FUNCTION_BLOCK StateMachine
VAR_INPUT
END_VAR
VAR_OUTPUT
END_VAR
VAR
	i : INT;
	State : States;
	TimerRotateDisc : TON;
	TimerLinearFW : TON;
	TimerGripperLower : TON;
	TimerGripperOpen : TON;
	TimerGripperClose: TON;
	TimerGripperLift: TON;
	TimerLinearBW : TON;
	Start: BOOL:=FALSE;
	CyclesCounter: CTU;
	TotalCyclesCounter : INT:=0;
	Reset : BOOL;
	NumberOfSlots : INT := 6;
	CylinderInDisc : ARRAY[1..6] OF BOOL := [FALSE, TRUE, TRUE, TRUE, TRUE, TRUE] ;
	Sensor: BOOL:= CylinderInDisc[4];
	PutCylinderInSlot6 : BOOL;
END_VAR

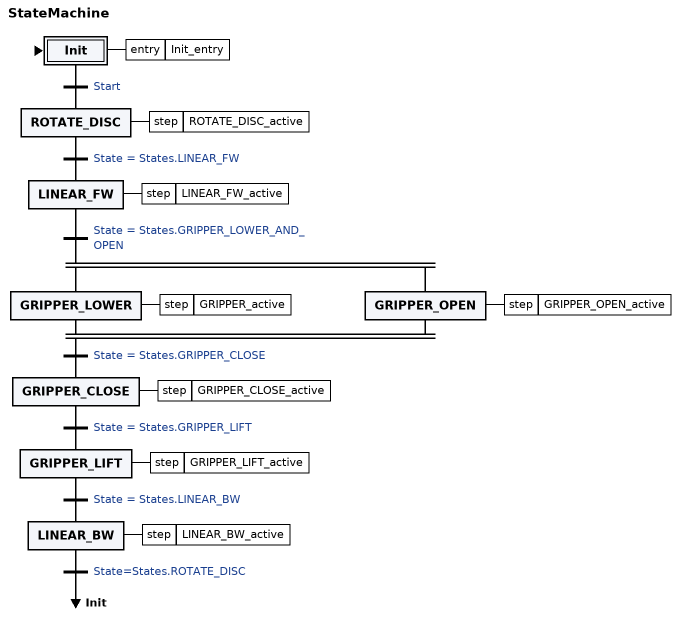
INITIAL_STEP Init:
    Init_entry(P1);  // entry action
END_STEP
TRANSITION FROM Init TO ROTATE_DISC
    := Start;
END_TRANSITION
STEP ROTATE_DISC:
    ROTATE_DISC_active(N);  // step action
END_STEP
TRANSITION FROM ROTATE_DISC TO LINEAR_FW
    := State = States.LINEAR_FW;
END_TRANSITION
STEP LINEAR_FW:
    LINEAR_FW_active(N);  // step action
END_STEP
TRANSITION FROM LINEAR_FW TO (GRIPPER_LOWER, GRIPPER_OPEN)
    := State = States.GRIPPER_LOWER_AND_OPEN;
END_TRANSITION
STEP GRIPPER_LOWER:
    GRIPPER_active(N);  // step action
END_STEP
STEP GRIPPER_OPEN:
    GRIPPER_OPEN_active(N);  // step action
END_STEP
TRANSITION FROM (GRIPPER_LOWER, GRIPPER_OPEN) TO GRIPPER_CLOSE
    := State = States.GRIPPER_CLOSE;
END_TRANSITION
STEP GRIPPER_CLOSE:
    GRIPPER_CLOSE_active(N);  // step action
END_STEP
TRANSITION FROM GRIPPER_CLOSE TO GRIPPER_LIFT
    := State = States.GRIPPER_LIFT;
END_TRANSITION
STEP GRIPPER_LIFT:
    GRIPPER_LIFT_active(N);  // step action
END_STEP
TRANSITION FROM GRIPPER_LIFT TO LINEAR_BW
    := State = States.LINEAR_BW;
END_TRANSITION
STEP LINEAR_BW:
    LINEAR_BW_active(N);  // step action
END_STEP
TRANSITION FROM LINEAR_BW TO Init
    := State=States.ROTATE_DISC;
END_TRANSITION

ACTION GRIPPER_active:
TimerGripperLower(IN:=TRUE, PT:=T#5S);
IF TimerGripperLower.Q THEN
	State := States.GRIPPER_CLOSE;
END_IF
END_ACTION

ACTION GRIPPER_CLOSE_active:
TimerGripperClose(IN:=TRUE, PT:=T#1S);
IF TimerGripperClose.Q THEN
	State := States.GRIPPER_LIFT;
END_IF
END_ACTION

ACTION GRIPPER_LIFT_active:
TimerGripperLift(IN:=TRUE, PT:=T#5S);
IF TimerGripperLift.Q THEN
	CylinderInDisc[1] := FALSE;
	State := States.LINEAR_BW;
END_IF
END_ACTION

ACTION GRIPPER_OPEN_active:
TimerGripperOpen(IN:=TRUE, PT:=T#1S);
END_ACTION

ACTION Init_entry:
Sensor := CylinderInDisc[4];

TimerRotateDisc(IN:=FALSE);
TimerLinearFW(IN:=FALSE);
TimerGripperLower(IN:=FALSE);
TimerGripperOpen(IN:=FALSE);
TimerGripperClose(IN:=FALSE);
TimerGripperLift(IN:=FALSE);
TimerLinearBW(IN:=FALSE);
Reset := CyclesCounter.Q;
CyclesCounter(CU:=state = States.ROTATE_DISC, RESET := Reset, PV:=INT_TO_WORD(NumberOfSlots));
END_ACTION

ACTION LINEAR_BW_active:
TimerLinearBW(IN:=TRUE, PT:=T#2S);
IF TimerLinearBW.Q THEN
	State := States.ROTATE_DISC;
END_IF
END_ACTION

ACTION LINEAR_FW_active:
TimerLinearFW(IN:=TRUE, PT:=T#2S);
IF TimerLinearFW.Q THEN
	State := States.GRIPPER_LOWER_AND_OPEN;
END_IF
END_ACTION

ACTION ROTATE_DISC_active:
TimerRotateDisc(IN:=TRUE, PT:=T#2S);

IF TimerRotateDisc.Q THEN
	TimerRotateDisc(IN:=FALSE);
	FOR i:=1 TO 5 BY 1 DO
		CylinderInDisc[i] := CylinderInDisc[i+1];
	END_FOR;
	CylinderInDisc[6] := PutCylinderInSlot6;
	IF CylinderInDisc[1] THEN
		State := States.LINEAR_FW;
	END_IF	
END_IF
END_ACTION

END_FUNCTION_BLOCK

(* stored: Version 1.1.0.1, ProductVersion 3.1.4024.12
   POU StateMachine: Id {90ec7814-8409-473f-9bb8-82d15f76498a}, SpecialFunc None
   Action GRIPPER_active: Id {12b64b9a-ca2e-4622-9620-65a67211656e}
   Action GRIPPER_CLOSE_active: Id {d691e21a-f8c1-4a63-8118-7801ba5c32fe}
   Action GRIPPER_LIFT_active: Id {4cd9cfc3-9895-41ad-abcb-f725e0d1d34a}
   Action GRIPPER_OPEN_active: Id {4fe590ed-dd1f-4566-b062-3ce9048b6aaf}
   Action Init_entry: Id {f8394b6a-6890-42bc-b48d-484abeb66bcb}
   Action LINEAR_BW_active: Id {04b344ae-3198-4f12-b7a5-389db0f028f0}
   Action LINEAR_FW_active: Id {c6f886f3-66c7-48bf-a531-e24bbdd03a9a}
   Action ROTATE_DISC_active: Id {0c13a474-856b-411f-9f0d-bd90afbbad44} *)
